# EPICS alarm handler configuration: epics/epics_alh/alarms_list_ScalerDAQ.alhConfig
GROUP NULL ScalerDAQ
